// TwinCAT 3 PLC project
// project tree:
//   POUs/ alg_x.TcPOU, alg_g_a_x.TcPOU, alg_g_z.TcPOU, alg_g_z2.TcPOU, alg_g_w_w.TcPOU, alg_g_w_W2.TcPOU, alg_g_a_X2.TcPOU, MAIN.TcPOU
//   DUTs/ STATE.TcDUT
//   GVLs/ TIMERS.TcGVL (not stored)

// ---- DUTs/STATE.TcDUT
TYPE STATE:
    STRUCT
        curTime: LREAL;
    END_STRUCT
END_TYPE

// ---- POUs/alg_x.TcPOU

      FUNCTION alg_x: LREAL
VAR_INPUT
    state: STATE;
END_VAR


        alg_x := state.curTime;

END_FUNCTION

// ---- POUs/alg_g_a_x.TcPOU
FUNCTION alg_g_a_x: LREAL
VAR_INPUT
    state: STATE;
END_VAR

alg_g_a_x := state.curTime;

END_FUNCTION

// ---- POUs/alg_g_z.TcPOU
FUNCTION alg_g_z: LREAL
VAR_INPUT
    state: STATE;
END_VAR

alg_g_z := state.curTime;

END_FUNCTION

// ---- POUs/alg_g_z2.TcPOU

      FUNCTION alg_g_z2: LREAL
VAR_INPUT
    state: STATE;
END_VAR


        alg_g_z2 := state.curTime;

END_FUNCTION

// ---- POUs/alg_g_w_w.TcPOU

      FUNCTION alg_g_w_w: LREAL
VAR_INPUT
    state: STATE;
END_VAR


        alg_g_w_w := state.curTime;

END_FUNCTION

// ---- POUs/alg_g_w_W2.TcPOU

      FUNCTION alg_g_w_W2: LREAL
VAR_INPUT
    state: STATE;
END_VAR


        alg_g_w_W2 := state.curTime;

END_FUNCTION

// ---- POUs/alg_g_a_X2.TcPOU
FUNCTION alg_g_a_X2: LREAL
VAR_INPUT
    state: STATE;
END_VAR

alg_g_a_X2 := state.curTime;

END_FUNCTION

// ---- POUs/MAIN.TcPOU
PROGRAM MAIN
VAR_OUTPUT
    timerValue0: TIME;
    timerValue1: TIME;
END_VAR
VAR
    cnt: LINT;
    first: BOOL := TRUE;
    curTimerValue: TIME;
    state0: STATE;
    curTime: LREAL;
    loopsKilled: LINT;
END_VAR
VAR_TEMP
    lastTimerValue: TIME;
    curDeltaTime: TIME;
    curDeltaSecs: LREAL;
    state1: STATE;
    progress: BOOL;
    loopCount: INT;
END_VAR


// Handle 'time' and cycle time.
cnt := cnt + 1;

timer0(IN := curTimer = 0, PT := T#1D);
timer1(IN := curTimer = 1, PT := T#1D);
timerValue0 := timer0.ET;
timerValue1 := timer1.ET;

lastTimerValue := curTimerValue;
IF curTimer = 0 THEN
    curTimerValue := timerValue0;
ELSE
    curTimerValue := timerValue1;
END_IF;
curDeltaTime := curTimerValue - lastTimerValue;
curDeltaSecs := TIME_TO_LREAL(curDeltaTime) / 1000;
curTime := curTime + curDeltaSecs;

IF cnt MOD 10 = 0 THEN
    curTimer := 1 - curTimer;
    curTimerValue := T#0S;
    timer0(IN := curTimer = 0, PT := T#1D);
    timer1(IN := curTimer = 1, PT := T#1D);
    timerValue0 := timer0.ET;
    timerValue1 := timer1.ET;
END_IF;

IF first THEN
    first := FALSE;

    // Initialize state variables for initial state.
ELSE
    // Update continuous variables for time delay.

    state0.curTime := curTime;
END_IF;

// Event loop.
WHILE TRUE DO
    progress := FALSE;

    // Done with events?
    IF NOT progress THEN
        EXIT;
    END_IF;

    // Protect against events that are always enabled.
    loopCount := loopCount + 1;
    IF loopCount >= 100 THEN
        loopsKilled := loopsKilled + 1;
        EXIT;
    END_IF;
END_WHILE;

END_PROGRAM
